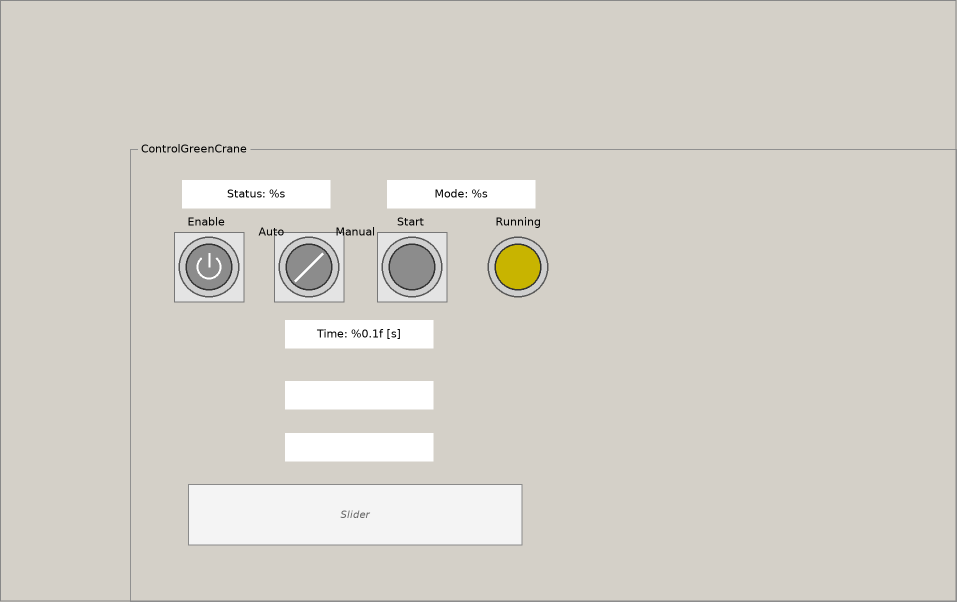
VISUALIZATION Visualization  // 957x602
    GroupBox (130,141 827x461), "ControlGreenCrane"
        Slider (58,343 334x61), scale 0..0.5
        PowerSwitch (44,91 70x70), variable: G_ControllerGreenCrane.bEnable, behaviour: TOGGLE, style: Switch-PowerSwitch-Gray
        RotarySwitch (144,91 70x70), variable: G_ControllerGreenCrane.bMode, behaviour: TOGGLE, style: Switch-RotarySwitch-Gray
        PushSwitch (247,91 70x70), variable: G_ControllerGreenCrane.bStart, behaviour: TOGGLE, style: Switch-PushSwitch-Gray
        Lamp1 (353,91 70x70), variable: G_ControllerGreenCrane.bLamp, style: Lamp-Lamp1-Yellow
        Textfield (51,38 150x30), "Status: %s", text variable: G_ControllerGreenCrane.eStatus
        Textfield (256,38 150x30), "Mode: %s", text variable: G_ControllerGreenCrane.eMode
        Textfield (154,291 150x30)
        Textfield (154,239 150x30)
        Textfield (154,178 150x30), "Time: %0.1f [s]", text variable: G_ControllerGreenCrane.fTimer
        Label (90,80 103x22), "Auto"
        Label (337,70 103x22), "Running"
        Label (229,70 103x22), "Start"
        Label (25,70 103x22), "Enable"
        Label (174,80 103x22), "Manual"
END_VISUALIZATION

(* stored: Version 1.1.0.1, ProductVersion 3.1.4024.12
   Visu Visualization: Id {e85578d3-e09c-4ff1-bfd6-4e76197ae7c9} *)
